FUNCTION SPLITTING_WORD_INTO_BYTES
  (* Standard: 61499-1; Description: Copyright (c) 2024 HR Agrartechnik GmbH This program and the accompanying materials are made available under the terms of the Eclipse Public License 2.0 which is available at https://www.eclipse.org/legal/epl-2.0/ SPDX-License-Identifier: EPL-2.0 *)
  (* Version 1.0, 2024-02-22, franz *)
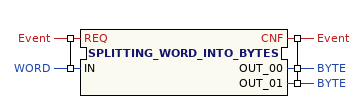
  EVENT_INPUT
    REQ WITH IN; (* Normal Execution Request *)
  END_EVENT
  EVENT_OUTPUT
    CNF WITH OUT_00, OUT_01; (* Execution Confirmation *)
  END_EVENT
  VAR_INPUT
    IN : WORD; (* WORD Input *)
  END_VAR
  VAR_OUTPUT
    OUT_00 : BYTE; (* BYTE 00 *)
    OUT_01 : BYTE; (* BYTE 01 *)
  END_VAR
  BODY IN ST:
FUNCTION SPLITTING_WORD_INTO_BYTES

VAR_INPUT
	IN : WORD;    // WORD Input
END_VAR

VAR_OUTPUT
	OUT_00 : BYTE;    // BYTE 00
	OUT_01 : BYTE;    // BYTE 01
END_VAR

(* this Function extracts the 2 BYTE from a word *)
OUT_00 := WORD_TO_BYTE(SHR(IN AND WORD_BYTE_00, SHFT_BYTE_00));
OUT_01 := WORD_TO_BYTE(SHR(IN AND WORD_BYTE_01, SHFT_BYTE_01));

END_FUNCTION
  END_BODY
END_FUNCTION
